// TIA Portal project "第二节课置位复位" (V15.1)

(* hardware
DEVICE "S7-1200 station_1"  S7-1200 Station
   slot 0: "Rack_0"  S7-1200 Rack  Rack  V1.0
   slot 1: "PLC_1"  CPU 1212C DC/DC/DC  6ES7 212-1AE40-0XB0  V4.2
*)

// ===== PLC "PLC_1"  CPU 1212C DC/DC/DC =====

VAR_GLOBAL   // PLC tag table "io"
   "开始" AT %I0.0 : Bool;
   "标志" AT %M0.0 : Bool;
   "复位" AT %I0.1 : Bool;
   "电机" AT %Q0.0 : Bool;
   "Tag_1" AT %I0.2 : Bool;
   "Tag_2" AT %M0.1 : Bool;
   "Tag_3" AT %I0.3 : Bool;
   "Tag_4" AT %M0.2 : Bool;
END_VAR

ORGANIZATION_BLOCK "Main"   // OB1, LAD, ProgramCycle
TITLE = "Main Program Sweep (Cycle)"
{ S7_Optimized_Access := 'TRUE' }
VERSION : 0.1
   VAR_INPUT
      Initial_Call : Bool;   // Initial call of this OB
      Remanence : Bool;   // =True, if remanent data are available
   END_VAR
BEGIN

REGION Network 1
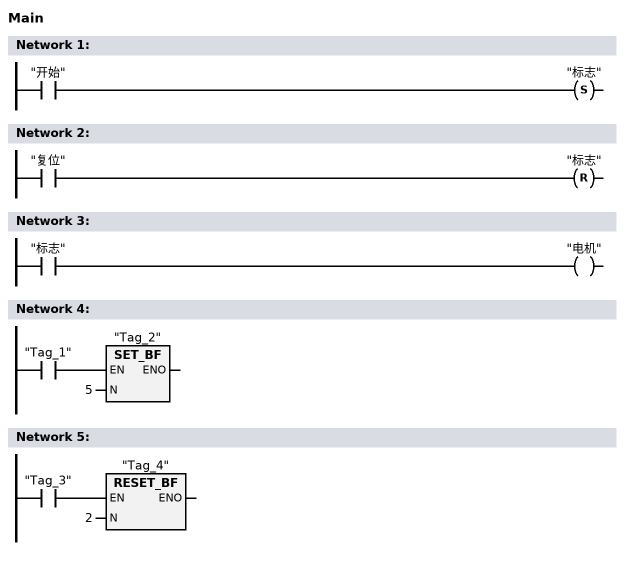
   RUNG wire#powerrail
      Contact( "开始" )
      S_Coil( "标志" )
   END_RUNG
   // the same network as SCL:
   IF "开始" THEN "标志" := TRUE; END_IF;
END_REGION

REGION Network 2
   RUNG wire#powerrail
      Contact( "复位" )
      R_Coil( "标志" )
   END_RUNG
   // the same network as SCL:
   IF "复位" THEN "标志" := FALSE; END_IF;
END_REGION

REGION Network 3
   RUNG wire#powerrail
      Contact( "标志" )
      Coil( "电机" )
   END_RUNG
   // the same network as SCL:
   "电机" := "标志";
END_REGION

REGION Network 4
   // no SCL statement known for SBitfield: written as a call
   IF "Tag_1" THEN SET_BF(operand := "Tag_2", n := 5); END_IF;
END_REGION

REGION Network 5
   // no SCL statement known for RBitfield: written as a call
   IF "Tag_3" THEN RESET_BF(operand := "Tag_4", n := 2); END_IF;
END_REGION
END_ORGANIZATION_BLOCK